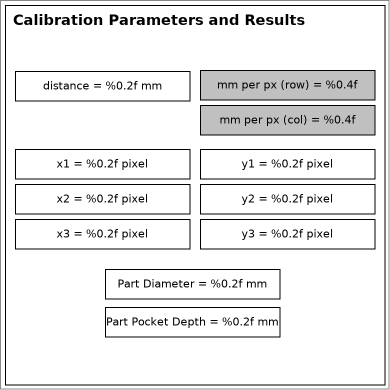
VISUALIZATION Manual_Camera_Calibration  // 390x390
    Rectangle (5,5 380x380)
    Rectangle (15,149 175x30), "x1 = %0.2f pixel", text variable: MAIN.fbSlitter.Camera._patternX1
    Rectangle (200,149 175x30), "y1 = %0.2f pixel", text variable: MAIN.fbSlitter.Camera._patternY1
    Rectangle (15,184 175x30), "x2 = %0.2f pixel", text variable: MAIN.fbSlitter.Camera._patternX2
    Rectangle (200,184 175x30), "y2 = %0.2f pixel", text variable: MAIN.fbSlitter.Camera._patternY2
    Rectangle (15,71 175x30), "distance = %0.2f mm", text variable: MAIN.fbSlitter.Camera._hmiParameters.calibrationDistance
        OnMouseClick: write MAIN.fbSlitter.Camera._hmiParameters.calibrationDistance via Default, title 'Load Position X'
    Rectangle (200,70 175x30), "mm per px (row) = %0.4f", text variable: MAIN.fbSlitter.Camera._parameters.pitchRow
    Label (10,5 297x30), "Calibration Parameters and Results"
    Rectangle (105,269 175x30), "Part Diameter = %0.2f mm", text variable: MAIN.fbSlitter.Camera._tubeParameters.Diameter
    Rectangle (105,307 175x30), "Part Pocket Depth = %0.2f mm", text variable: MAIN.fbSlitter.Camera._tubeParameters.DepthOfPocket
    Rectangle (15,219 175x30), "x3 = %0.2f pixel", text variable: MAIN.fbSlitter.Camera._patternX3
    Rectangle (200,219 175x30), "y3 = %0.2f pixel", text variable: MAIN.fbSlitter.Camera._patternY3
    Rectangle (200,105 175x30), "mm per px (col) = %0.4f", text variable: MAIN.fbSlitter.Camera._parameters.pitchColumn
END_VISUALIZATION

(* stored: Version 1.1.0.1, ProductVersion 3.1.4024.9
   Visu Manual_Camera_Calibration: Id {f696f724-c2d3-4631-9b51-d2eb37b6df6f} *)
